// TwinCAT 3 PLC project TrafficLight
// ProgramVersion: 3.1.4024.0
// libraries:
//   Tc2_Standard, * (Beckhoff Automation GmbH)
//   Tc2_System, * (Beckhoff Automation GmbH)
//   Tc3_Module, * (Beckhoff Automation GmbH)
//   VisuDialogs, * (System)
// project tree:
//   / GlobalTextList.TcGTLO, PlcTask.TcTTO, Visualization Manager.TcVMO (not stored)
//   POUs/ FB_Blinker.TcPOU, FB_TrafficLight.TcPOU, MAIN.TcPOU
//   VISUs/ Visualization.TcVIS
// real-time tasks:
//   TASK PlcTask: cycle T#10ms, priority 20, ADS port 350
// I/O:
//   DEVICE Device 2 (EtherCAT) (disabled), AmsNetId 10.0.20.81.3.1
//     Term 1 (EK1100) [EK1100 EtherCAT Coupler (2A E-Bus)]
//       Term 2 (EL1014) [EL1014 4Ch. Dig. Input 24V, 10µs]
//       Term 3 (EL2004) [EL2004 4Ch. Dig. Output 24V, 0.5A]
//       Term 4 (EL9011) [EL9011 End Terminal]
// variable links:
//   TrafficLight/TrafficLight Instance <-> Device 2 (EtherCAT)/Term 1 (EK1100)/Term 2 (EL1014)
//     PlcTask Inputs/MAIN.fbTrafficLight.bIsBlinkPressed <-> Channel 3/Input
//     PlcTask Inputs/MAIN.fbTrafficLight.bIsStartPressed <-> Channel 1/Input
//     PlcTask Inputs/MAIN.fbTrafficLight.bIsStopPressed <-> Channel 2/Input
//   TrafficLight/TrafficLight Instance <-> Device 2 (EtherCAT)/Term 1 (EK1100)/Term 3 (EL2004)
//     PlcTask Outputs/MAIN.fbTrafficLight.bTurnGreenLightOn <-> Channel 3/Output
//     PlcTask Outputs/MAIN.fbTrafficLight.bTurnRedLightOn <-> Channel 1/Output
//     PlcTask Outputs/MAIN.fbTrafficLight.bTurnYellowLightOn <-> Channel 2/Output

CONFIGURATION TrafficLight
    RESOURCE PLC ON TwinCAT3
        TASK PlcTask(INTERVAL := T#10ms, PRIORITY := 20);
        PROGRAM MAIN WITH PlcTask : MAIN;
    END_RESOURCE
END_CONFIGURATION

// ---- POUs/MAIN.TcPOU
PROGRAM MAIN
VAR
	bIsStartPressed : BOOL;
	bIsStopPressed : BOOL;
	bIsBlinkPressed : BOOL;

	fbTrafficLight : FB_TrafficLight;
	
	dwRedTimeOn : DWORD := 8000;
	
	dwRedAndYellowTimeOn : DWORD := 1000;
	
	dwGreenTimeOn : DWORD := 5000;
	
	dwGreenBlinkingDuration : DWORD := 2000;
	dwGreenBlinkingTimeOn : DWORD := 250;
	dwGreenBlinkingTimeOff : DWORD := 100;
	
	dwYellowTimeOn : DWORD := 1000;
	
	dwYellowBlinkingTimeOn : DWORD := 250;
	dwYellowBlinkingTimeOff : DWORD := 100;
END_VAR

fbTrafficLight(bIsStartPressed := bIsStartPressed, bIsStopPressed := bIsStopPressed, bIsBlinkPressed := bIsBlinkPressed,
			   dwRedTimeOn := dwRedTimeOn,
			   dwRedAndYellowTimeOn := dwRedAndYellowTimeOn, 
			   dwGreenTimeOn := dwGreenTimeOn,
			   dwGreenBlinkingDuration := dwGreenBlinkingDuration, dwGreenBlinkingTimeOn := dwGreenBlinkingTimeOn, dwGreenBlinkingTimeOff := dwGreenBlinkingTimeOff,
			   dwYellowTimeOn := dwYellowTimeOn,
			   dwYellowBlinkingTimeOn := dwYellowBlinkingTimeOn, dwYellowBlinkingTimeOff := dwYellowBlinkingTimeOff,);		   
			   
//// For connection with hardware
//fbTrafficLight(dwRedTimeOn := dwRedTimeOn,
//			   dwRedAndYellowTimeOn := dwRedAndYellowTimeOn, 
//			   dwGreenTimeOn := dwGreenTimeOn,
//			   dwGreenBlinkingDuration := dwGreenBlinkingDuration, dwGreenBlinkingTimeOn := dwGreenBlinkingTimeOn, dwGreenBlinkingTimeOff := dwGreenBlinkingTimeOff,
//			   dwYellowTimeOn := dwYellowTimeOn,
//			   dwYellowBlinkingTimeOn := dwYellowBlinkingTimeOn, dwYellowBlinkingTimeOff := dwYellowBlinkingTimeOff,);

END_PROGRAM

// ---- POUs/FB_TrafficLight.TcPOU
FUNCTION_BLOCK FB_TrafficLight
VAR_INPUT
	bIsStartPressed AT %I* : BOOL;
	bIsStopPressed AT %I* : BOOL;
	bIsBlinkPressed AT %I* : BOOL;

	dwRedTimeOn : DWORD;	// Duration for red light on

	dwRedAndYellowTimeOn : DWORD;	

	dwGreenTimeOn : DWORD;
	
	dwGreenBlinkingDuration : DWORD;
	dwGreenBlinkingTimeOn : DWORD;
	dwGreenBlinkingTimeOff : DWORD;
	
	dwYellowTimeOn : DWORD;
	
	dwYellowBlinkingTimeOn : DWORD;
	dwYellowBlinkingTimeOff : DWORD;
END_VAR
VAR_OUTPUT
	bTurnGreenLightOn AT %Q* : BOOL;
	bTurnYellowLightOn AT %Q* : BOOL;
	bTurnRedLightOn AT %Q* : BOOL;
END_VAR
VAR
	fbRedTimerOn : TON;
	
	fbRedAndYellowTimerOn : TON;
	
	fbGreenTimerOn : TON;
	
	fbGreenBlinker : FB_Blinker;
	fbGreenBlinkingTimerOn : TON;
	fbGreenBlinkingTimerOff : TON;
	
	fbYellowTimerOn : TON;
	
	fbYellowBlinker : FB_Blinker;
	
	(* 0 - Yellow blinking; 50 - Initialization; 100 - Red; 
	200 - Red + Yellow; 300 - Green; 400 - Yellow*)
	eLightOrder : INT := 0;
	
	// In order to showcase the remaining time (countdown)
	dwGreenTimeRemaining : DWORD;
	dwRedTimeRemaining : DWORD;
END_VAR

CASE eLightOrder OF	
	0:	// Yellow blinking
		bTurnGreenLightOn := FALSE;
        bTurnYellowLightOn := FALSE;
        bTurnRedLightOn := FALSE;
		
		 // Check if the start button is pressed to start the traffic light 
        IF bIsStartPressed THEN
            eLightOrder := 100;
		
		// Go to initialization if stop button is pressed, if not turn on yellow blinker
		ELSIF bIsStopPressed THEN
        	eLightOrder := 50;
		ELSE
			fbYellowBlinker(dwTimeOn := dwYellowBlinkingTimeOn, dwTimeOff := dwYellowBlinkingTimeOff, bLight => bTurnYellowLightOn);
		END_IF	
	
	50:			
		// Initialization
		bTurnGreenLightOn := FALSE;
        bTurnYellowLightOn := FALSE;
        bTurnRedLightOn := FALSE;
		
		// Reseting all timers
		fbRedTimerOn(IN := FALSE);
		fbRedAndYellowTimerOn(IN := FALSE);
		fbGreenTimerOn(IN := FALSE);
		fbGreenBlinkingTimerOn(IN := FALSE);
		fbGreenBlinkingTimerOff(IN := FALSE);
		fbYellowTimerOn(IN := FALSE);
        
        // Check if the start button is pressed to start the traffic light 
        IF bIsStartPressed THEN
            eLightOrder := 100;
        END_IF
		
		// Check if the blink button is pressed to start the yellow light blinking
		IF bIsBlinkPressed THEN
            eLightOrder := 0;
        END_IF

	100:	// Red
		IF bIsStopPressed THEN
            eLightOrder := 50;
		ELSIF bIsBlinkPressed THEN
            eLightOrder := 0;
        ELSE
			bTurnGreenLightOn := FALSE;
			bTurnYellowLightOn := FALSE;
			bTurnRedLightOn := TRUE;
			
			// Start red light timer
			fbRedTimerOn(IN := TRUE, PT := DWORD_TO_TIME(dwRedTimeOn));
			dwRedTimeRemaining := TIME_TO_DWORD((fbRedTimerOn.PT - fbRedTimerOn.ET) / 1000);
			
			// Transition to next state when timer elapses
			IF fbRedTimerOn.Q THEN
				fbRedTimerOn(IN := FALSE);
				eLightOrder := 200;
			END_IF
		END_IF
	
	200:	// Red + Yellow
		IF bIsStopPressed THEN
            eLightOrder := 50;
		ELSIF bIsBlinkPressed THEN
            eLightOrder := 0;
        ELSE
			bTurnGreenLightOn := FALSE;
			bTurnYellowLightOn := TRUE;
			bTurnRedLightOn := TRUE;
			
			// Start red and yellow light timer
			fbRedAndYellowTimerOn(IN := TRUE, PT := DWORD_TO_TIME(dwRedAndYellowTimeOn));
			
			// Transition to next state when timer elapses
			IF fbRedAndYellowTimerOn.Q THEN
				fbRedAndYellowTimerOn(IN := FALSE);
				eLightOrder := 300;
			END_IF
		END_IF
	
	300:	// Green
		IF bIsStopPressed THEN
            eLightOrder := 50;
		ELSIF bIsBlinkPressed THEN
            eLightOrder := 0;
        ELSE
			bTurnGreenLightOn := TRUE;
			bTurnYellowLightOn := FALSE;
			bTurnRedLightOn := FALSE;
			
			// Start green light timer
			fbGreenTimerOn(IN := TRUE, PT := DWORD_TO_TIME(dwGreenTimeOn));
			dwGreenTimeRemaining := TIME_TO_DWORD((fbGreenTimerOn.PT - fbGreenTimerOn.ET) / 1000);
			
			// Transition to next state when timer elapses
			IF fbGreenTimerOn.Q THEN
				fbGreenTimerOn(IN := FALSE);
				eLightOrder := 400;
			END_IF
		END_IF
		
	400:	// Yellow
		IF bIsStopPressed THEN
            eLightOrder := 50;
		ELSIF bIsBlinkPressed THEN
            eLightOrder := 0;
        ELSE
			bTurnGreenLightOn := FALSE;
			bTurnYellowLightOn := TRUE;
			bTurnRedLightOn := FALSE;
			
			// Start yellow light timer
			fbYellowTimerOn(IN := TRUE, PT := DWORD_TO_TIME(dwYellowTimeOn));
			
			// Transition to next state when timer elapses
			IF fbYellowTimerOn.Q THEN
				fbYellowTimerOn(IN := FALSE);
				eLightOrder := 100;
			END_IF
		END_IF
ELSE	// There is some fault - yellow blinking
	eLightOrder := 0;
END_CASE

END_FUNCTION_BLOCK

// ---- POUs/FB_Blinker.TcPOU
FUNCTION_BLOCK FB_Blinker
VAR_INPUT
	dwTimeOn : DWORD;
	dwTimeOff : DWORD;
END_VAR
VAR_OUTPUT
	bLight : BOOL;	// Determines whether the light will be ON or OFF
END_VAR
VAR
	fbTimerOn : TON;
	fbTimerOff : TON;
	fbStartTrigger : R_TRIG;
	
	eCurrentPhase : INT := 10;	// 10 - ON, 20 - OFF
	
	bIsBlinking : bool;
END_VAR

CASE eCurrentPhase OF
    10:	// ON
        fbTimerOn(IN := TRUE, PT := DWORD_TO_TIME(dwTimeOn));
        IF fbTimerOn.Q THEN
            fbTimerOn(IN := FALSE); // Reset the on timer
            eCurrentPhase := 20;  // Move to the off phase
        END_IF
        bLight := TRUE;

    20:	// OFF
        fbTimerOff(IN := TRUE, PT := DWORD_TO_TIME(dwTimeOff));
        IF fbTimerOff.Q THEN
            fbTimerOff(IN := FALSE); // Reset the off timer
            eCurrentPhase := 10;  // Move to the On phase
        END_IF
        bLight := FALSE;
		
ELSE
	fbTimerOn(IN := FALSE);
    fbTimerOff(IN := FALSE);
    bLight := FALSE;
END_CASE

END_FUNCTION_BLOCK

// ---- GlobalTextList.TcGTLO
TEXTLIST GlobalTextList
  709 = '%s'
  214 = 'BLINK'
  426 = 'Change green blinking duration'
  66 = 'Change green blinking off time'
  570 = 'Change green blinking on time'
  71 = 'Change green light time'
  620 = 'Change red and yellow time'
  886 = 'Change red light time'
  366 = 'Change yellow blinking off time'
  240 = 'Change yellow blinking on time'
  118 = 'Change yellow blinking time'
  470 = 'Change yellow light time'
  349 = 'Green blinker time'
  232 = 'Green light time'
  605 = 'Pokazhi vreme %s'
  55 = 'Red light time'
  981 = 'START'
  692 = 'START / STOP'
  242 = 'STOP'
  251 = 'Time on: %s'
  607 = 'Time ON: %s'
  936 = 'YELLOW BLINKING'
  521 = 'Yellow light time'
END_TEXTLIST

// ---- VISUs/Visualization.TcVIS
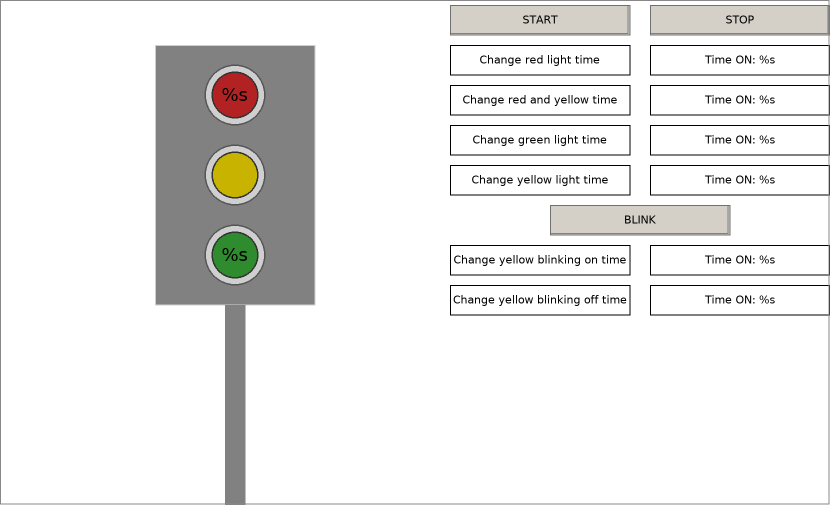
VISUALIZATION Visualization  // 830x505
    Rectangle (155,45 160x260)
    Lamp1 (200,60 70x70), variable: MAIN.fbTrafficLight.bTurnRedLightOn, style: Lamp-Lamp1-Red
    Lamp1 (200,140 70x70), variable: MAIN.fbTrafficLight.bTurnYellowLightOn, style: Lamp-Lamp1-Yellow
    Lamp1 (200,220 70x70), variable: MAIN.fbTrafficLight.bTurnGreenLightOn, style: Lamp-Lamp1-Green
    Rectangle (225,305 20x200)
    Rectangle (450,45 180x30), "Change red light time"
        OnMouseClick: write MAIN.dwRedTimeOn via Default
    Rectangle (450,85 180x30), "Change red and yellow time"
        OnMouseClick: write MAIN.dwRedAndYellowTimeOn via Default
    Rectangle (450,125 180x30), "Change green light time"
        OnMouseClick: write MAIN.dwGreenTimeOn via Default
    Rectangle (450,165 180x30), "Change yellow light time"
        OnMouseClick: write MAIN.dwYellowTimeOn via Default
    Rectangle (220,80 30x30), "%s", text variable: MAIN.fbTrafficLight.dwRedTimeRemaining, invisible if: NOT MAIN.fbTrafficLight.bTurnRedLightOn OR MAIN.fbTrafficLight.bTurnYellowLightOn
    Rectangle (220,240 30x30), "%s", text variable: MAIN.fbTrafficLight.dwGreenTimeRemaining, invisible if: NOT (MAIN.fbTrafficLight.eLightOrder = 300)
    Rectangle (450,245 180x30), "Change yellow blinking on time"
        OnMouseClick: write MAIN.dwYellowBlinkingTimeOn via Default
    Rectangle (450,285 180x30), "Change yellow blinking off time"
        OnMouseClick: write MAIN.dwYellowBlinkingTimeOff via Default
    Rectangle (650,45 180x30), "Time ON: %s", text variable: MAIN.fbTrafficLight.fbRedTimerOn.ET
    Rectangle (650,85 180x30), "Time ON: %s", text variable: MAIN.fbTrafficLight.fbRedAndYellowTimerOn.ET
    Rectangle (650,125 180x30), "Time ON: %s", text variable: MAIN.fbTrafficLight.fbGreenTimerOn.ET
    Rectangle (650,165 180x30), "Time ON: %s", text variable: MAIN.fbTrafficLight.fbYellowTimerOn.ET
    Rectangle (650,245 180x30), "Time ON: %s", text variable: MAIN.fbTrafficLight.fbYellowBlinker.fbTimerOn.ET
    Rectangle (650,285 180x30), "Time ON: %s", text variable: MAIN.fbTrafficLight.fbYellowBlinker.fbTimerOff.ET
    Button (450,5 180x30), "START"
        tap MAIN.bIsStartPressed
    Button (650,5 180x30), "STOP"
        tap MAIN.bIsStopPressed
    Button (550,205 180x30), "BLINK"
        tap main.bIsBlinkPressed
END_VISUALIZATION
